TYPE ST_PlcEventDef :
STRUCT
	bEventSignal	:BOOL;
	nEventID		:INT;
	nEventType	:INT:=1;	(*1:Alarm , 2:Warning , *)
END_STRUCT
END_TYPE

(* stored: Version 1.1.0.1, ProductVersion 3.1.4024.6
   DUT ST_PlcEventDef: Id {7a56770a-55ac-4cd3-87df-a9ea5750993b} *)
